// TIA Portal V17 export
// export: Created 2024-06-14T09:53:11.099488Z, ExportSetting WithDefaults, DisplayName Totally Integrated Automation Portal, DisplayVersion V17, DisplayName TIA Portal Openness, DisplayVersion V17, DisplayName TIA Portal Version Control Interface, DisplayVersion V17, DisplayName Simotion SCOUT TIA, DisplayVersion 5.4.3.0, DisplayName SINAMICS Startdrive Advanced, DisplayVersion V17 SP1 Update 1, DisplayName SINAMICS Startdrive G110M, G120, G120C, G120D, G120P, G115D, DisplayVersion V17 SP1 Update 1, DisplayName SINAMICS Startdrive G130, G150, S120, S150, SINAMICS MV, S210, DisplayVersion V17 SP1 Update 1, DisplayName STEP 7 Professional, DisplayVersion V17, DisplayName STEP 7 Safety, DisplayVersion V17, DisplayName WinCC Professional, DisplayVersion V17
DATA_BLOCK "LPG_Check_scale_FB_DB"   // DB48
VERSION : 0.1
// stored: AutoNumber true, DBAccessibleFromOPCUA true, InstanceOfName LPG_Check_scale_FB, InstanceOfType FB
"LPG_Check_scale_FB"
   // VAR_INPUT
   //    INxCylinder_In_Pos : Bool;
   //    INxAuto_Start_Seq : Bool;
   //    INxMan_Start_Seq : Bool;
   //    INxStop_Sequence : Bool;
   //    INtStart_TImeout_Time : DInt;
   //    INxReset_Sequence : Bool;
   //    INxCylinder_Type : Int;
   //    INrTare_Entry_SP : Real;
   //    DOWN_CONVEYOR : Bool;
   //    data_delete : Bool;
   // END_VAR
   // VAR_OUTPUT
   //    OutuFilled_Data : Array[1..10] of Real;
   //    OutxDomestic_Cylinder : Bool;
   //    OutxCommercial_Cylinder : Bool;
   //    OutxStart_Timeout : Bool;
   //    OutxTare_Entry_Error : Bool;
   //    Outx_Filling_Error : Bool;
   //    Outx_Tare_Value_Error : Bool;
   //    Cycle_Started : Bool;
   //    OutiStep_No : Int;
   //    OUTiResult : Int;
   //    Gross_Weight : Real;
   //    Net_Wieght : Real;
   //    Tare_Weight : Real;
   //    OUT_Decision : Int;
   // END_VAR
   // VAR_IN_OUT
   //    Modbus_Master_DB : "MOD_MASTER_DATA_1";
   // END_VAR
   // VAR
   //    TRIG : Array[1..25] of Bool;
   //    STEP_NO : Int;
   //    Step_Timer { S7_SetPoint := 'True'} : Array[1..15] of IEC_TIMER;
   //    Domestic_Cylinder { S7_SetPoint := 'True'} : Bool;
   //    Commercial_Cylinder : Bool;
   //    Cyl_Done { S7_SetPoint := 'True'} : TOF_TIME;
   //    Tare_Enrty_Extn { S7_SetPoint := 'True'} : TOF_TIME;
   //    Start_Timeout_Err { S7_SetPoint := 'True'} : TON_TIME;
   //    Tare_Entry_Timer { S7_SetPoint := 'True'} : TON_TIME;
   //    Filled_Gross : Real;
   //    Filled_Net : Real;
   //    Punched_Tare : Real;
   //    Test_Seq : Int;
   //    RESULT : Bool;
   //    IEC_Timer_0_Instance { S7_SetPoint := 'True'} : TOF_TIME;
   //    Gross { S7_SetPoint := 'True'} : Real;
   //    gross_diff : Real;
   //    pass : Bool;
   //    Decision : Word;
   //    IEC_Timer_0_Instance_1 { S7_SetPoint := 'True'} : TON_TIME;
   //    fill { S7_SetPoint := 'True'} : TON_TIME;
   //    ALL_FILL_DONE : Bool;
   // END_VAR
   // VAR RETAIN
   //    cycle_start { S7_SetPoint := 'True'} : CTU_INT;
   // END_VAR
BEGIN
END_DATA_BLOCK
